Universal Robots PolyScope program: demo str weld.urp

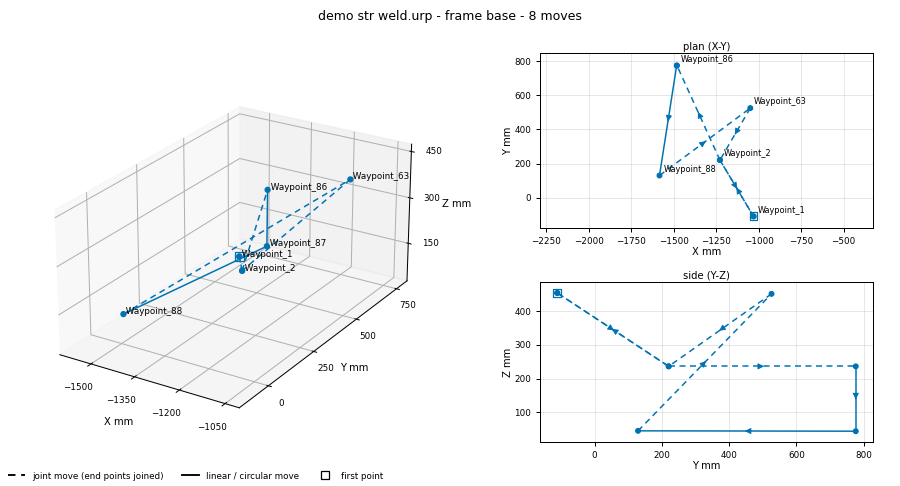
[picture p0: tool path of demo str weld.urp in frame base, 8 of 8 moves have a stored position in this frame; points joined in program order, loops and branches not executed]
Program demo str weld (installation=default directory=/programs createdIn=5.21.3 lastSavedIn=5.21.3 robotSerialNumber=20246801938)
Calibrated DH parameters: a=[-0.000071, -0.790281, -0.600694, 0.000061, -0.000039, 0]; d=[0.236272, 604.465945, 132.116513, -736.382239, 0.159268, 0.154005]; alpha=[1.570254, -0.000567, 0.000559, 1.571709, -1.56999, 0]; deltaTheta=[0, -0.409357, 7.293326, -0.600784, -0.000001, -0.000001]
InitVariablesNode
Robot Program (runOnlyOnce=true)
  Set NoAction tcp=pretend_welder
  MoveJ speed 60 deg/s, acceleration 80 deg/s^2 (useActiveTCP=true optimoveEnabled=false optiMoveSpeed=0.3 optiMoveAcceleration=0.09) feature=Base
    SafeHome (positionOptionType=SPEED_AND_ACCELERATION speed=1.047198 acceleration=1.396263 nextMotionTime=2)
    Waypoint Waypoint_1: TCP in base x=-1030.165 y=-110.755 z=454.213 mm, rx=1.6835 ry=-2.4103 rz=-0.3725 rad; joints [-20.283, -69.554, 90.976, 63.422, -0.136, -102.51] deg; TCP offset x=-9.5 y=-328 z=105.73 mm, rx=1.2092 ry=-1.2092 rz=1.2092 rad
    Waypoint Waypoint_2: TCP in base x=-1227.598 y=220.265 z=236.167 mm, rx=0.2832 ry=3.09 rz=0.0697 rad; joints [-20.205, -68.009, 92.689, -22.783, 80.38, -3.042] deg
    SuppressedNode
      Waypoint Waypoint_59: TCP in base x=-1227.598 y=220.265 z=517.582 mm, rx=0.2832 ry=3.09 rz=0.0697 rad; joints [-20.196, -72.607, 76.22, -1.718, 80.38, -3.031] deg
  MoveJ speed 60 deg/s, acceleration 80 deg/s^2 (useActiveTCP=true optimoveEnabled=false optiMoveSpeed=0.3 optiMoveAcceleration=0.09) feature=Base
    SuppressedNode
      Waypoint Waypoint_1: TCP in base x=-1030.165 y=-110.755 z=454.213 mm, rx=1.6835 ry=-2.4103 rz=-0.3725 rad; joints [-20.283, -69.554, 90.976, 63.422, -0.136, -102.51] deg
    SuppressedNode
      Waypoint Waypoint_2: TCP in base x=-1227.598 y=220.265 z=236.167 mm, rx=0.2832 ry=3.09 rz=0.0697 rad; joints [-20.205, -68.009, 92.689, -22.783, 80.38, -3.042] deg
    SuppressedNode
      Waypoint Waypoint_3: TCP in base x=-1118.347 y=-386.264 z=236.167 mm, rx=0.2832 ry=3.09 rz=0.0697 rad; joints [15.781, -68.529, 93.461, -22.819, 116.345, -1.79] deg
    SuppressedNode
      Waypoint Waypoint_7: TCP in base x=-1160.376 y=-386.264 z=236.167 mm, rx=0.2832 ry=3.09 rz=0.0697 rad; joints [15.132, -66.213, 89.988, -21.674, 115.695, -1.818] deg
    SuppressedNode
      Waypoint Waypoint_10: TCP in base x=-1209.873 y=-386.264 z=236.167 mm, rx=-0.3182 ry=-3.1015 rz=-0.0802 rad; joints [15.165, -64.461, 88.659, -26.025, 116.89, -3.591] deg
    SuppressedNode
      Waypoint Waypoint_13: TCP in base x=-1272.267 y=-386.264 z=236.167 mm, rx=-0.3182 ry=-3.1015 rz=-0.0802 rad; joints [14.313, -60.941, 83.063, -23.936, 116.038, -3.562] deg
    SuppressedNode
      Waypoint Waypoint_16: TCP in base x=-1330.142 y=-308.947 z=236.167 mm, rx=-0.3182 ry=-3.1015 rz=-0.0802 rad; joints [9.786, -59.392, 80.532, -22.896, 111.512, -3.408] deg
    SuppressedNode
      Waypoint aironly1: TCP in base x=-1365.007 y=-308.947 z=236.167 mm, rx=-0.3182 ry=-3.1015 rz=-0.0802 rad; joints [9.492, -57.272, 77.008, -21.489, 111.218, -3.399] deg
    SuppressedNode
      Waypoint Waypoint_20: TCP in base x=-1417.271 y=-308.947 z=236.167 mm, rx=-0.3182 ry=-3.1015 rz=-0.0802 rad; joints [9.082, -53.986, 71.407, -19.169, 110.807, -3.387] deg
    SuppressedNode
      Waypoint Waypoint_23: TCP in base x=-1480.309 y=-308.947 z=236.167 mm, rx=-0.3182 ry=-3.1015 rz=-0.0802 rad; joints [8.632, -49.786, 64.02, -15.978, 110.356, -3.373] deg
    SuppressedNode
      Waypoint Waypoint_26: TCP in base x=-1520.922 y=-308.947 z=236.167 mm, rx=-0.3182 ry=-3.1015 rz=-0.0802 rad; joints [8.365, -46.89, 58.787, -13.638, 110.087, -3.365] deg
    SuppressedNode
      Waypoint Waypoint_29: TCP in base x=-1577.729 y=-291.057 z=236.167 mm, rx=-0.3182 ry=-3.1015 rz=-0.0802 rad; joints [7.27, -42.895, 51.39, -10.225, 108.99, -3.33] deg
    SuppressedNode
      Waypoint Waypoint_32: TCP in base x=-1648.288 y=-245.474 z=236.167 mm, rx=-0.3182 ry=-3.1015 rz=-0.0802 rad; joints [5.081, -37.626, 41.338, -5.422, 106.799, -3.262] deg
    SuppressedNode
      Waypoint Waypoint_35: TCP in base x=-1589.386 y=-277.501 z=243.673 mm, rx=-0.057 ry=-3.1131 rz=-0.0768 rad; joints [4.821, -44.028, 52.909, -10.537, 96.927, -2.966] deg
    SuppressedNode
      Waypoint Waypoint_38: TCP in base x=-987.212 y=220.265 z=-2.697 mm, rx=-0.2872 ry=-3.1249 rz=-0.0133 rad; joints [-27.869, -71.721, 123.355, -51.945, 72.696, -0.347] deg
    SuppressedNode
      Waypoint Waypoint_40: TCP in base x=-1008.917 y=39.093 z=-94.513 mm, rx=-0.2669 ry=-3.1267 rz=-0.0132 rad; joints [-14.12, -65.442, 125.083, -59.932, 85.7, -0.424] deg
    SuppressedNode
      Waypoint Waypoint_42: TCP in base x=-964.636 y=395.957 z=-76.673 mm, rx=-0.2872 ry=-3.1249 rz=-0.0133 rad; joints [-40.131, -65.269, 122.082, -57.156, 60.434, -0.278] deg
    SuppressedNode
      Waypoint Waypoint_44: TCP in base x=-1073.002 y=19.222 z=-79.792 mm, rx=-0.2519 ry=-3.128 rz=-0.0133 rad; joints [-11.766, -63.634, 119.38, -56.027, 87.506, -0.437] deg
    SuppressedNode
      Waypoint Waypoint_47: TCP in base x=-966.075 y=73.096 z=-108.967 mm, rx=-0.1617 ry=-3.1342 rz=-0.0142 rad; joints [-19.175, -66.279, 129.103, -63.09, 76.795, -0.431] deg
    SuppressedNode
      Waypoint Waypoint_50: TCP in base x=-1016.839 y=73.096 z=-108.967 mm, rx=-0.1617 ry=-3.1342 rz=-0.0142 rad; joints [-17.869, -64.201, 124.85, -60.913, 78.101, -0.437] deg
    SuppressedNode
      Waypoint Waypoint_53: TCP in base x=-1068.513 y=73.096 z=-108.967 mm, rx=-0.1617 ry=-3.1342 rz=-0.0142 rad; joints [-16.711, -62.061, 120.455, -58.657, 79.259, -0.442] deg
    SuppressedNode
      Waypoint Waypoint_56: TCP in base x=-1020.608 y=73.096 z=-108.967 mm, rx=-0.1617 ry=-3.1342 rz=-0.0142 rad; joints [-17.779, -64.046, 124.532, -60.75, 78.191, -0.437] deg
    SuppressedNode
      Waypoint Waypoint_60: TCP in base x=-1489.675 y=380.494 z=425.287 mm, rx=0.2336 ry=3.0935 rz=0.0688 rad; joints [-23.255, -50.293, 48.601, 3.711, 75.49, -3.169] deg
    SuppressedNode
      Waypoint Waypoint_65: TCP in base x=-1256.292 y=6.475 z=12.774 mm, rx=0.208 ry=3.1308 rz=0.0037 rad; joints [-9.369, -59.685, 100.822, -40.971, 88.295, -0.127] deg; TCP offset x=-9.5 y=-328 z=105 mm, rx=1.2092 ry=-1.2092 rz=1.2092 rad
    SuppressedNode
      Waypoint Waypoint_68: TCP in base x=-1394.879 y=124.829 z=28.16 mm, rx=0.2793 ry=3.1252 rz=0.0035 rad; joints [-13.538, -52.645, 86.413, -33.604, 86.738, -0.132] deg
    SuppressedNode
      Waypoint Waypoint_73: TCP in base x=-1440.255 y=178.159 z=50.313 mm, rx=0.2577 ry=3.1271 rz=0.0036 rad; joints [-15.712, -50.589, 80.526, -29.774, 83.77, -0.14] deg
    SuppressedNode
      Waypoint Waypoint_74: TCP in base x=-1587.602 y=209.495 z=50.809 mm, rx=0.2577 ry=3.1271 rz=0.0036 rad; joints [-15.293, -40.972, 62.077, -20.941, 84.184, -0.139] deg
    SuppressedNode
      Waypoint Waypoint_77: TCP in base x=-1350.226 y=220.265 z=152.903 mm, rx=0.1939 ry=3.1027 rz=-0.0205 rad; joints [-19.745, -58.234, 84.308, -24.159, 77.465, 0.254] deg
    SuppressedNode
      Waypoint Waypoint_80: TCP in base x=-1271.202 y=220.265 z=152.903 mm, rx=0.1955 ry=3.125 rz=-0.0185 rad; joints [-21.335, -63.377, 93.308, -29.327, 75.884, 0.523] deg
    SuppressedNode
      Waypoint Waypoint_83: TCP in base x=-1465.492 y=220.265 z=236.167 mm, rx=0.2578 ry=3.128 rz=-0.0047 rad; joints [-17.383, -53.706, 70.17, -16.328, 82.098, 0.171] deg
    Waypoint Waypoint_86: TCP in base x=-1480.462 y=776.092 z=236.167 mm, rx=0.2578 ry=3.128 rz=-0.0047 rad; joints [-38.663, -37.36, 40.1, -2.598, 60.81, 0.113] deg
  MoveL speed 100 mm/s, acceleration 1200 mm/s^2 (useActiveTCP=true optimoveEnabled=false optiMoveSpeed=0.3 optiMoveAcceleration=0.09) feature=Base
    SuppressedNode
      Waypoint Waypoint_4: TCP in base x=-1118.347 y=-386.264 z=131.592 mm, rx=0.2832 ry=3.09 rz=0.0697 rad; joints [15.778, -65.168, 97.71, -30.431, 116.343, -1.797] deg; TCP offset x=-9.5 y=-328 z=105.73 mm, rx=1.2092 ry=-1.2092 rz=1.2092 rad
    SuppressedNode
      Waypoint Waypoint_6: TCP in base x=-1118.231 y=-386.375 z=138.305 mm, rx=0.2834 ry=3.0952 rz=0.0665 rad; joints [15.78, -65.53, 97.763, -30.435, 116.329, -1.785] deg
    SuppressedNode
      Waypoint Waypoint_8: TCP in base x=-1171.679 y=-386.264 z=140.683 mm, rx=0.2832 ry=3.09 rz=0.0697 rad; joints [14.962, -62.717, 92.928, -28.116, 115.528, -1.83] deg
    SuppressedNode
      Waypoint Waypoint_11: TCP in base x=-1218.84 y=-386.264 z=141.877 mm, rx=-0.3182 ry=-3.1015 rz=-0.0802 rad; joints [15.033, -61.094, 91.598, -32.332, 116.76, -3.592] deg
    SuppressedNode
      Waypoint Waypoint_14: TCP in base x=-1272.267 y=-386.264 z=141.352 mm, rx=-0.3182 ry=-3.1015 rz=-0.0802 rad; joints [14.31, -58.23, 86.815, -30.402, 116.037, -3.567] deg
    SuppressedNode
      Waypoint Waypoint_17: TCP in base x=-1311.178 y=-308.947 z=135.898 mm, rx=-0.3182 ry=-3.1015 rz=-0.0802 rad; joints [9.95, -57.664, 86.333, -30.428, 111.679, -3.419] deg
    SuppressedNode
      Waypoint Waypoint_19: TCP in base x=-1311.353 y=-308.947 z=145.167 mm, rx=-0.3182 ry=-3.1015 rz=-0.0802 rad; joints [9.949, -57.948, 85.991, -29.802, 111.677, -3.418] deg
    SuppressedNode
      Waypoint aironly2: TCP in base x=-1365.007 y=-308.947 z=146.214 mm, rx=-0.3182 ry=-3.1015 rz=-0.0802 rad; joints [9.489, -54.916, 80.643, -27.482, 111.217, -3.404] deg
    SuppressedNode
      Waypoint Waypoint_21: TCP in base x=-1414.861 y=-308.947 z=146.661 mm, rx=-0.3182 ry=-3.1015 rz=-0.0802 rad; joints [9.098, -51.97, 75.377, -25.157, 110.824, -3.391] deg
    SuppressedNode
      Waypoint Waypoint_24: TCP in base x=-1463.949 y=-308.947 z=145.333 mm, rx=-0.3182 ry=-3.1015 rz=-0.0802 rad; joints [8.742, -48.886, 69.895, -22.756, 110.468, -3.38] deg
    SuppressedNode
      Waypoint Waypoint_27: TCP in base x=-1512.175 y=-308.947 z=151.315 mm, rx=-0.3182 ry=-3.1015 rz=-0.0802 rad; joints [8.419, -45.854, 63.788, -19.677, 110.143, -3.37] deg
    SuppressedNode
      Waypoint Waypoint_30: TCP in base x=-1576.574 y=-291.057 z=149.826 mm, rx=-0.3182 ry=-3.1015 rz=-0.0802 rad; joints [7.273, -41.58, 55.832, -15.984, 108.996, -3.334] deg
    SuppressedNode
      Waypoint Waypoint_33: TCP in base x=-1630.659 y=-245.474 z=148.621 mm, rx=-0.1755 ry=-3.1105 rz=-0.0784 rad; joints [4.178, -39.136, 51.224, -13.757, 100.644, -3.078] deg
    SuppressedNode
      Waypoint Waypoint_36: TCP in base x=-1595.127 y=-277.501 z=158.706 mm, rx=-0.057 ry=-3.1131 rz=-0.0768 rad; joints [4.798, -42.195, 56.286, -15.747, 96.906, -2.968] deg
    SuppressedNode
      Waypoint Waypoint_39: TCP in base x=-1008.917 y=39.093 z=-149.869 mm, rx=-0.2669 ry=-3.1267 rz=-0.0132 rad; joints [-14.123, -61.447, 125.875, -64.719, 85.696, -0.429] deg
    SuppressedNode
      Waypoint Waypoint_43: TCP in base x=-965.936 y=395.957 z=-145.567 mm, rx=-0.2872 ry=-3.1249 rz=-0.0133 rad; joints [-40.072, -60.527, 123.017, -62.829, 60.493, -0.285] deg
    SuppressedNode
      Waypoint Waypoint_45: TCP in base x=-1070.759 y=19 z=-148.949 mm, rx=-0.2519 ry=-3.128 rz=-0.0133 rad; joints [-11.786, -59.194, 120.56, -61.647, 87.485, -0.443] deg
    SuppressedNode
      Waypoint Waypoint_48: TCP in base x=-964.364 y=73.096 z=-154.996 mm, rx=-0.1617 ry=-3.1342 rz=-0.0142 rad; joints [-19.225, -62.748, 129.889, -67.406, 76.744, -0.435] deg
    SuppressedNode
      Waypoint Waypoint_51: TCP in base x=-1020.114 y=74.442 z=-152.898 mm, rx=-0.161 ry=-3.1216 rz=-0.0194 rad; joints [-17.895, -60.878, 125.707, -65.842, 78.071, -0.44] deg
    SuppressedNode
      Waypoint Waypoint_54: TCP in base x=-1068.989 y=73.096 z=-154.088 mm, rx=-0.1617 ry=-3.1342 rz=-0.0142 rad; joints [-16.704, -59.013, 120.982, -62.231, 79.266, -0.446] deg
    SuppressedNode
      Waypoint Waypoint_57: TCP in base x=-1017.692 y=74.382 z=-152.109 mm, rx=-0.1612 ry=-3.1222 rz=-0.0191 rad; joints [-17.946, -61.026, 125.874, -65.82, 78.025, -0.44] deg
    SuppressedNode
      Waypoint Waypoint_61: TCP in base x=-1489.588 y=379.777 z=323.956 mm, rx=0.2336 ry=3.0935 rz=0.0688 rad; joints [-23.23, -49.99, 56.054, -4.044, 75.518, -3.17] deg
    SuppressedNode
      Waypoint Waypoint_64: TCP in base x=-1481.572 y=434.13 z=331.518 mm, rx=0.2336 ry=3.0935 rz=0.0688 rad; joints [-25.602, -49.491, 54.574, -3.041, 73.147, -3.258] deg
    SuppressedNode
      Waypoint Waypoint_66: TCP in base x=-1254.156 y=6.475 z=-46.113 mm, rx=0.208 ry=3.1308 rz=0.0037 rad; joints [-9.392, -57.056, 102.313, -45.092, 88.273, -0.131] deg; TCP offset x=-9.5 y=-328 z=105 mm, rx=1.2092 ry=-1.2092 rz=1.2092 rad
    SuppressedNode
      Waypoint Waypoint_69: TCP in base x=-1394.879 y=124.829 z=-56.508 mm, rx=0.2793 ry=3.1252 rz=0.0035 rad; joints [-13.541, -49.302, 88.254, -38.788, 86.736, -0.136] deg
    SuppressedNode
      Waypoint Waypoint_72: TCP in base x=-1440.255 y=178.159 z=-60.937 mm, rx=0.2577 ry=3.1271 rz=0.0036 rad; joints [-15.715, -46.488, 83.059, -36.406, 83.767, -0.145] deg
    SuppressedNode
      Waypoint Waypoint_75: TCP in base x=-1587.983 y=209.495 z=-53.031 mm, rx=0.2577 ry=3.1271 rz=0.0036 rad; joints [-15.291, -37.805, 64.687, -26.717, 84.187, -0.144] deg
    SuppressedNode
      Waypoint Waypoint_78: TCP in base x=-1345.209 y=220.265 z=49.508 mm, rx=-0.1951 ry=-3.1289 rz=0.0245 rad; joints [-20.071, -55.833, 90.449, -34.995, 77.128, 1.029] deg
    SuppressedNode
      Waypoint Waypoint_81: TCP in base x=-1270.494 y=220.99 z=38.34 mm, rx=-0.196 ry=-3.1349 rz=0.013 rad; joints [-21.392, -59.318, 97.642, -38.382, 75.826, 0.516] deg
    SuppressedNode
      Waypoint Waypoint_84: TCP in base x=-1484.183 y=98.372 z=40.786 mm, rx=0.2578 ry=3.128 rz=-0.0047 rad; joints [-11.585, -48.006, 76.527, -28.383, 87.899, 0.176] deg
    Waypoint Waypoint_87: TCP in base x=-1481.957 y=776.092 z=43.475 mm, rx=0.2578 ry=3.128 rz=-0.0047 rad; joints [-38.631, -34.399, 49.642, -15.098, 60.846, 0.106] deg
  Folder turn ext on
    URCap WireTank Serial (WireTank Serial, WireTank, LLC) dataModel(NODE_TITLE=Serial Bridge uR1, Command=[252,82,49], QUERY=false, OUTPUT_ENTRY=Static, byte_array=true, Variable(key=OUTPUT_VARIABLE, variable(name=HwResp)))
    URCap WireTank Serial (WireTank Serial, WireTank, LLC) dataModel(NODE_TITLE=Serial Bridge uR1, Command=[252,82,49], byte_array=true, OUTPUT_ENTRY=Static, QUERY=false, Variable(key=OUTPUT_VARIABLE, variable=HwResp))
    Wait Sleep waitTime=1
    SuppressedNode
      Script: turn_extrusion_on()
    Set DigitalOutput pin=digital_out[0]; digitalValue=1
  Wait Sleep waitTime=1
  MoveL speed 10 mm/s, acceleration 1200 mm/s^2 (useActiveTCP=true optimoveEnabled=false optiMoveSpeed=0.3 optiMoveAcceleration=0.09) feature=Base
    SuppressedNode
      Waypoint Waypoint_5: TCP in base x=-1022.03 y=88.8 z=129.642 mm, rx=0.2832 ry=3.09 rz=0.0697 rad; joints [-16.194, -77.207, 115.563, -36.474, 84.391, -2.911] deg; TCP offset x=-9.5 y=-328 z=105.73 mm, rx=1.2092 ry=-1.2092 rz=1.2092 rad
    SuppressedNode
      Waypoint Waypoint_9: TCP in base x=-1069.353 y=129.9 z=143.412 mm, rx=0.2832 ry=3.09 rz=0.0697 rad; joints [-18.053, -74.88, 111.041, -34.272, 82.533, -2.972] deg
    SuppressedNode
      Waypoint Waypoint_12: TCP in base x=-1062.423 y=416.712 z=141.359 mm, rx=-0.3182 ry=-3.1015 rz=-0.0802 rad; joints [-36.035, -72.334, 109.197, -38.685, 65.714, -2.016] deg
    SuppressedNode
      Waypoint Waypoint_15: TCP in base x=-1125.045 y=359.119 z=137.922 mm, rx=-0.3182 ry=-3.1015 rz=-0.0802 rad; joints [-30.592, -69.948, 106.012, -37.815, 71.155, -2.199] deg
    SuppressedNode
      Waypoint Waypoint_18: TCP in base x=-1193.677 y=324.269 z=140.17 mm, rx=-0.3182 ry=-3.1015 rz=-0.0802 rad; joints [-26.629, -66.815, 100.994, -35.891, 75.116, -2.325] deg
    SuppressedNode
      Waypoint aironly3: TCP in base x=-1252.116 y=291.882 z=146.428 mm, rx=-0.3175 ry=-3.0928 rz=-0.0841 rad; joints [-23.442, -64.356, 96.74, -34.588, 78.297, -2.422] deg
    SuppressedNode
      Waypoint Waypoint_22: TCP in base x=-1284.956 y=387.801 z=148.559 mm, rx=-0.3182 ry=-3.1015 rz=-0.0802 rad; joints [-27.494, -61.035, 90.892, -31.576, 74.25, -2.299] deg
    SuppressedNode
      Waypoint Waypoint_25: TCP in base x=-1338.671 y=332.562 z=143.961 mm, rx=-0.3182 ry=-3.1015 rz=-0.0802 rad; joints [-23.594, -58.657, 87.309, -30.34, 78.148, -2.42] deg
    SuppressedNode
      Waypoint Waypoint_28: TCP in base x=-1382.953 y=322.31 z=144.2 mm, rx=-0.3182 ry=-3.1015 rz=-0.0802 rad; joints [-22.22, -56.205, 83.072, -28.546, 79.521, -2.461] deg
    SuppressedNode
      Waypoint Waypoint_31: TCP in base x=-1455.501 y=414.683 z=145.052 mm, rx=-0.3182 ry=-3.1015 rz=-0.0802 rad; joints [-24.923, -50.416, 72.709, -23.991, 76.817, -2.381] deg
    SuppressedNode
      Waypoint Waypoint_34: TCP in base x=-1535.127 y=406.733 z=146.561 mm, rx=-0.1755 ry=-3.1105 rz=-0.0784 rad; joints [-24.201, -45.339, 63.218, -19.616, 72.279, -2.24] deg
    SuppressedNode
      Waypoint Waypoint_37: TCP in base x=-1546.229 y=365.536 z=159.597 mm, rx=-0.057 ry=-3.1131 rz=-0.0768 rad; joints [-23.223, -45.495, 62.436, -18.718, 68.898, -2.13] deg
    SuppressedNode
      Waypoint Waypoint_41: TCP in base x=-935.469 y=635.881 z=-147.989 mm, rx=0.2263 ry=3.1319 rz=0.0049 rad; joints [-53.73, -56.038, 113.125, -57.064, 44.6, -0.192] deg
    SuppressedNode
      Waypoint Waypoint_46: TCP in base x=-1028.965 y=318.99 z=-150.456 mm, rx=-0.2353 ry=-3.1293 rz=-0.0133 rad; joints [-33.319, -59.018, 120.409, -61.705, 65.343, -0.326] deg
    SuppressedNode
      Waypoint Waypoint_49: TCP in base x=-924.132 y=611.05 z=-146.55 mm, rx=-0.1617 ry=-3.1342 rz=-0.0142 rad; joints [-53.867, -56.955, 115.146, -58.588, 42.103, -0.205] deg
    SuppressedNode
      Waypoint Waypoint_52: TCP in base x=-971.384 y=683.258 z=-149.074 mm, rx=-0.161 ry=-3.1216 rz=-0.0194 rad; joints [-54.294, -53.507, 108.335, -56.33, 41.678, 0.469] deg
    SuppressedNode
      Waypoint Waypoint_55: TCP in base x=-1019.488 y=723.134 z=-143.33 mm, rx=-0.1617 ry=-3.1342 rz=-0.0142 rad; joints [-53.246, -51.062, 101.769, -51.099, 42.723, -0.21] deg
    SuppressedNode
      Waypoint Waypoint_58: TCP in base x=-973.975 y=701.326 z=-149.834 mm, rx=-0.1612 ry=-3.1222 rz=-0.0191 rad; joints [-54.793, -52.876, 107.012, -55.592, 41.184, 0.451] deg
    SuppressedNode
      Waypoint Waypoint_62: TCP in base x=-1449.725 y=620.724 z=330.286 mm, rx=0.2336 ry=3.0935 rz=0.0688 rad; joints [-33.47, -46.347, 49.03, -0.537, 65.283, -3.566] deg
    SuppressedNode
      Waypoint Waypoint_67: TCP in base x=-1188.535 y=687.972 z=-44.736 mm, rx=0.1927 ry=3.1318 rz=0.0037 rad; joints [-44.849, -50.287, 89.016, -38.537, 52.254, -0.25] deg; TCP offset x=-9.5 y=-328 z=105 mm, rx=1.2092 ry=-1.2092 rz=1.2092 rad
    SuppressedNode
      Waypoint Waypoint_70: TCP in base x=-1299.115 y=817.148 z=-56.462 mm, rx=0.2577 ry=3.1271 rz=0.0036 rad; joints [-45.063, -40.773, 71.058, -30.095, 54.416, -0.241] deg
    SuppressedNode
      Waypoint Waypoint_71: TCP in base x=-1351.222 y=817.148 z=-54.87 mm, rx=0.2577 ry=3.1271 rz=0.0036 rad; joints [-43.463, -38.137, 65.529, -27.207, 56.015, -0.234] deg
    SuppressedNode
      Waypoint Waypoint_76: TCP in base x=-1499.222 y=843.63 z=-48.844 mm, rx=0.2577 ry=3.1271 rz=0.0036 rad; joints [-40.212, -27.718, 43.472, -15.573, 59.259, -0.222] deg
    SuppressedNode
      Waypoint Waypoint_79: TCP in base x=-1267.78 y=775.15 z=41.356 mm, rx=-0.1951 ry=-3.1289 rz=0.0245 rad; joints [-45.416, -46.907, 74.576, -28.151, 51.781, 1.236] deg
    SuppressedNode
      Waypoint Waypoint_82: TCP in base x=-1205.018 y=704.901 z=37.009 mm, rx=-0.196 ry=-3.1349 rz=0.013 rad; joints [-45.025, -52.175, 84.789, -32.698, 52.191, 0.547] deg
    SuppressedNode
      Waypoint Waypoint_85: TCP in base x=-1385.278 y=733.037 z=41.544 mm, rx=0.2578 ry=3.128 rz=-0.0047 rad; joints [-39.802, -42.264, 65.396, -22.986, 59.68, 0.103] deg
    Waypoint Waypoint_88: TCP in base x=-1583.023 y=129.317 z=44.575 mm, rx=0.2578 ry=3.128 rz=-0.0047 rad; joints [-12.04, -41.639, 63.915, -22.139, 87.441, 0.174] deg
  URCap WireTank Serial (WireTank Serial, WireTank, LLC) dataModel(QUERY=false, byte_array=true, NODE_TITLE=Serial Bridge uR0, Command=[252,82,48], OUTPUT_ENTRY=Static, Variable(key=OUTPUT_VARIABLE, variable(name=HwResp)))
  MoveL speed 250 mm/s, acceleration 1200 mm/s^2 (useActiveTCP=true optimoveEnabled=false optiMoveSpeed=0.3 optiMoveAcceleration=0.09) feature=Base
    MoveDirectionNode (selectedDirection=ZPlus)
      Until DISTANCE (allowActions=false deceleration=3 distanceNodeType=STOP) Distance=0.15; motionParameters(blendRadius=0)
  Set DigitalOutput pin=digital_out[0]; digitalValue=0
  MoveJ speed 60 deg/s, acceleration 80 deg/s^2 (useActiveTCP=true optimoveEnabled=false optiMoveSpeed=0.3 optiMoveAcceleration=0.09) feature=Base
    Waypoint Waypoint_63: TCP in base x=-1049.013 y=525.841 z=451.462 mm, rx=0.2463 ry=3.0924 rz=0.0692 rad; joints [-42.164, -76.681, 86.797, -7.814, 57.068, -3.935] deg; TCP offset x=-9.5 y=-328 z=105.73 mm, rx=1.2092 ry=-1.2092 rz=1.2092 rad
    Waypoint Waypoint_2: TCP in base x=-1227.598 y=220.265 z=236.167 mm, rx=0.2832 ry=3.09 rz=0.0697 rad; joints [-20.205, -68.009, 92.689, -22.783, 80.38, -3.042] deg
    Waypoint Waypoint_1: TCP in base x=-1030.165 y=-110.755 z=454.213 mm, rx=1.6835 ry=-2.4103 rz=-0.3725 rad; joints [-20.283, -69.554, 90.976, 63.422, -0.136, -102.51] deg
  SafeHome (positionOptionType=SPEED_AND_ACCELERATION speed=1.047198 acceleration=1.396263 nextMotionTime=2)
